// Checks if a character is a digit
FUNCTION F_IsDigit : BOOL
VAR_INPUT
	t_Char : T_Char;
END_VAR

F_IsDigit := t_Char >= '0' AND t_Char <= '9';

END_FUNCTION

(* stored: Version 1.1.0.1, ProductVersion 3.1.4024.4
   POU F_IsDigit: Id {096fc1e7-8253-4366-8b9d-f2db44130b22}, SpecialFunc None *)
